FUNCTION_BLOCK FB_05
VAR_INPUT
END_VAR
VAR_OUTPUT
END_VAR
VAR
END_VAR

END_FUNCTION_BLOCK

(* stored: Version 1.1.0.1, ProductVersion 3.1.4024.12
   POU FB_05: Id {daf9b826-0aea-4e1a-bddc-d3e3b8eb1b86}, SpecialFunc None *)
